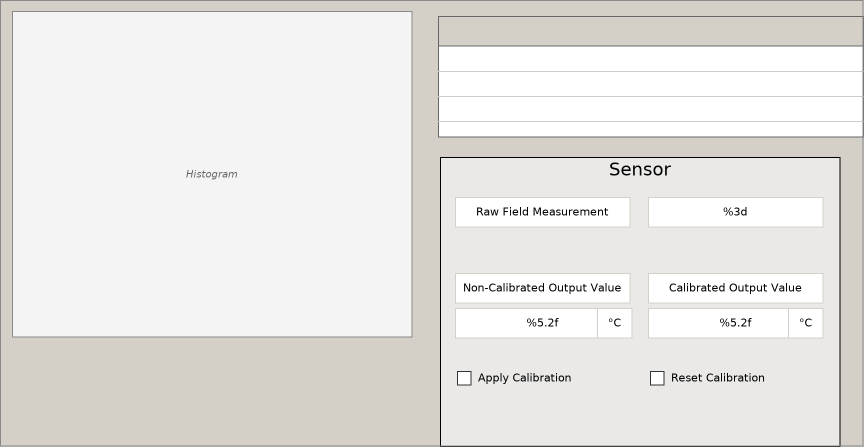
VISUALIZATION Visualization_Calibration_Screen  // 864x447
    RoundedRectangle (440,157 400x290), "Sensor"
    Histogram (12,11 400x326), scale format: %.1f, scale 0..100
        p518627256: °C
        p1518820177: Temperature_Transducer_A1_Calibration.Reference_Points
        p102497268: Temperature_Transducer_A1_Calibration.Reference_Points
        p788070771: ARRAY [1..Calibration_Points] OF REAL
    Textfield (455,308 175x30), "%5.2f", text variable: Temperature_Transducer_A1_Calibration.Sensor_Input_Value
    Textfield (455,273 175x30), "Non-Calibrated Output Value"
    Table (438,16 426x121), data array: Temperature_Transducer_A1_Calibration.Reference_Points
        p3854506369: Temperature_Transducer_A1_Calibration.Reference_Points[INDEX]
    Textfield (648,308 175x30), "%5.2f", text variable: Temperature_Transducer_A1_Calibration.Calibrated_Output_Value
    Textfield (648,273 175x30), "Calibrated Output Value"
    Checkbox (455,363 150x30), "Apply Calibration", variable: Temperature_Transducer_A1_Calibration.Start_Calibration
    Checkbox (648,363 150x30), "Reset Calibration", variable: Temperature_Transducer_A1_Calibration.Reset_Calibration
    Textfield (455,197 175x30), "Raw Field Measurement"
    Textfield (648,197 175x30), "%3d", text variable: Temperature_Transducer_A1.SimulatedRawValue
        OnMouseDown: write the text variable via Default, min 0, max 32768
    Textfield (788,308 35x30), "°C"
    Textfield (597,308 35x30), "°C"
END_VISUALIZATION

(* stored: Version 1.1.0.1, ProductVersion 3.1.4024.15
   Visu Visualization_Calibration_Screen: Id {e1009aa6-dbaa-46bc-8d53-fdedd1f1acb8} *)
